# EPICS autosave request: mrfApp/Db/evr-template-prescaler-to-pulse-gen.inc.req
$(P)$(R)Prescaler@PRESCALER_NUM@:MapTo:TrigPulseGen@PULSE_GEN_NUM@
